# B&R Automation Studio project SW_Shirokov_L2
Automation Studio 4.5.2.102

## Configuration SampleText

### Task classes (Cpu.sw)
```
Cyclic#1 (cycle 2000 us, tolerance 0 us):
  ncsdcctrl <- ncsdcctrl.prg
Cyclic#4:
  Program <- Program.prg
NcDataObjects: acp10etxen <- acp10etxen.dob, gAxis01a <- gAxis01obj.gAxis01a.dob, gAxis01i <- gAxis01obj.gAxis01i.dob
Libraries: Acp10sdc, sys_lib, Runtime, asstring, Library, Acp10man, Acp10par, NcGlobal, Acp10_MC, brsystem, AsBrStr
```

### Hardware
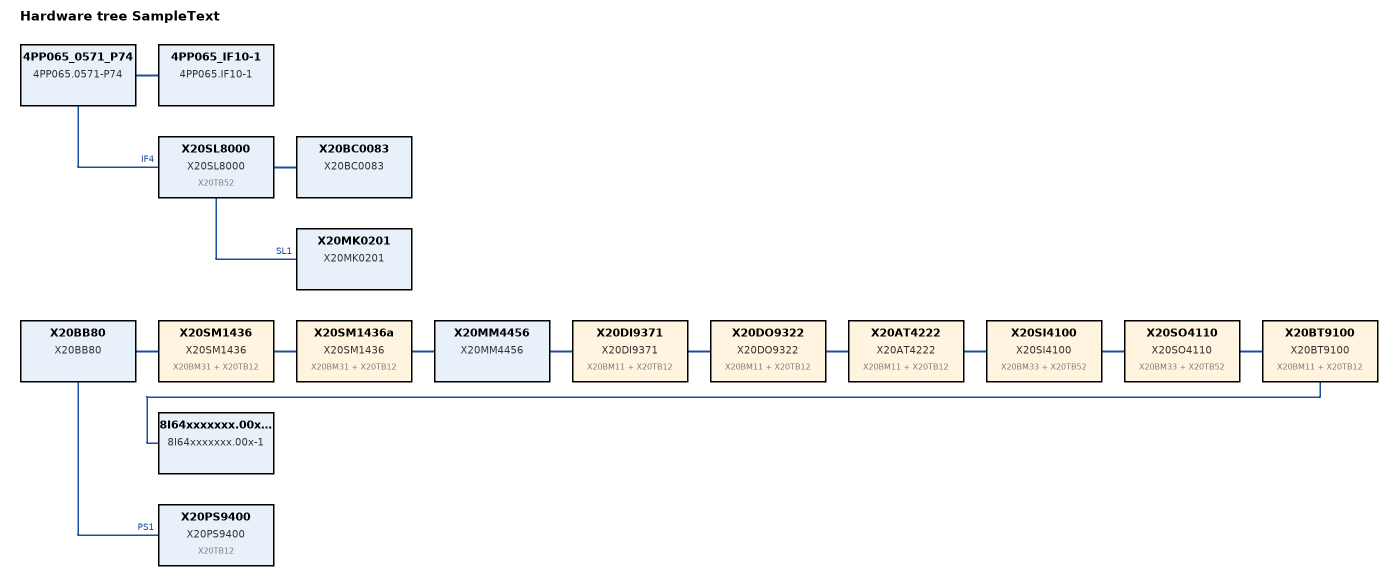
```
4PP065_0571_P74 : 4PP065.0571-P74 v1.1.2.0
  Connector IF5:
    ActivateDevice = 1
    Mode = Manual
    InternetAddress = 10.0.1.10
    SubnetMask = 255.255.255.0
  ConfigurationID = labBR
  TimerDeviceType = EPLX2X
  TimerDevice = 4PP065_0571_P74.IF4
  TaskClassIdleTime = 2000
  Cyclic1Duration = 2000
  Cyclic1Tolerance = 0
  Cyclic1Output = 1
4PP065_IF10-1 : 4PP065.IF10-1 v1.0.3.0  [SS -> 4PP065_0571_P74.SS1]
8I64xxxxxxx.00x-1 : 8I64xxxxxxx.00x-1 v1.3.9.1  [X2X1 -> X20BT9100.X2X1 [Cable Type=X2XCable, Length=10, Version=1.0.0.2]]
  packedETAD = packed
  packedETI = packed
  packedCMDD = packed
  packedCMI = packed
  ACC = 30
  UNS = 220
  NCR = 10
  NSP = 890
  COS = 64
  RSC = 33000
X20AT4222 : X20AT4222 v1.2.3.0  [SS1 -> X20TB12e.SS; SL -> X20BM11c.SL1]
X20BB80 : X20BB80 v1.0.2.0
X20BC0083 : X20BC0083 v2.14.0.0  [PLK1 -> X20SL8000.PLK2 (NodeNumber=2) [Cable Type=PowerlinkCable, Length=10, Version=1.0.0.2]; SL -> X20BB80.SL1]
X20BM11 : X20BM11 v1.0.0.1  [X2X1 -> X20BM33a.X2X2]
X20BM11a : X20BM11 v1.0.0.1  [X2X1 -> X20MM4456.X2X2]
X20BM11b : X20BM11 v1.0.0.1  [X2X1 -> X20BM11a.X2X2]
X20BM11c : X20BM11 v1.0.0.1  [X2X1 -> X20BM11b.X2X2]
X20BM31 : X20BM31 v1.0.0.1  [X2X1 -> X20BB80.IF1]
X20BM31a : X20BM31 v1.0.0.1  [X2X1 -> X20BM31.X2X2]
X20BM33 : X20BM33 v1.0.0.4  [X2X1 -> X20BM11c.X2X2]
X20BM33a : X20BM33 v1.0.0.4  [X2X1 -> X20BM33.X2X2]
X20BT9100 : X20BT9100 v1.0.3.0  [SS1 -> X20TB12f.SS; SL -> X20BM11.SL1]
X20DI9371 : X20DI9371 v1.0.2.0  [SS1 -> X20TB12c.SS; SL -> X20BM11a.SL1]
X20DO9322 : X20DO9322 v1.0.3.0  [SS1 -> X20TB12d.SS; SL -> X20BM11b.SL1]
X20MK0201 : X20MK0201 v1.0.0.0  [SL -> X20SL8000.SL1]
X20MM4456 : X20MM4456 v1.4.0.0  [X2X1 -> X20BM31a.X2X2]
X20PS9400 : X20PS9400 v1.0.2.4  [SS1 -> X20TB12.SS; PS -> X20BB80.PS1]
X20SI4100 : X20SI4100 v1.10.1.1  [SS1 -> X20TB52.SS; SL -> X20BM33.SL1]
X20SL8000 : X20SL8000 v1.6.5.1  [PLK1 -> 4PP065_0571_P74.IF4 (NodeNumber=1) [Cable Type=PowerlinkCable, Length=10, Version=1.0.0.2]; PLK2 -> X20BC0083.PLK1 (NodeNumber=1) [Cable Type=PowerlinkCable, Length=10, Version=1.0.0.2]; SS1 -> X20TB52b.SS]
  SafeProject = SafeLOGIC-1
X20SM1436 : X20SM1436 v2.3.0.0  [SS1 -> X20TB12a.SS; SL -> X20BM31.SL1]
X20SM1436a : X20SM1436 v2.3.0.0  [SS1 -> X20TB12b.SS; SL -> X20BM31a.SL1]
X20SO4110 : X20SO4110 v1.10.1.1  [SS1 -> X20TB52a.SS; SL -> X20BM33a.SL1]
  SafeModuleID = 3
X20TB12 : X20TB12 v1.0.0.0
X20TB12a : X20TB12 v1.0.0.0
X20TB12b : X20TB12 v1.0.0.0
X20TB12c : X20TB12 v1.0.0.0
X20TB12d : X20TB12 v1.0.0.0
X20TB12e : X20TB12 v1.0.0.0
X20TB12f : X20TB12 v1.0.0.0
X20TB52 : X20TB52 v1.0.0.1
X20TB52a : X20TB52 v1.0.0.1
X20TB52b : X20TB52 v1.0.0.1
```

### IoMap.iom - 4PP065_0571_P74/IoMap.iom
```iecst
VAR_CONFIG
	Cyclic#1.gAxis01_DrvIf.iLifeCnt AT %IB."8I64xxxxxxx.00x-1".SDC_LifeCnt;
	Cyclic#1.gAxis01_DrvIf.iDrvOK AT %IX."8I64xxxxxxx.00x-1".ETAD_Input_Bool_02;
	Cyclic#1.gAxis01_DrvIf.oSetTime AT %QW."8I64xxxxxxx.00x-1".SDC_SetTime;
	Cyclic#1.gAxis01_DiDoIf.iLifeCntDriveReady AT %IB."8I64xxxxxxx.00x-1".SDC_LifeCnt;
	Cyclic#1.gAxis01_DiDoIf.iLifeCntDriveEnable AT %IB."8I64xxxxxxx.00x-1".SDC_LifeCnt;
	Cyclic#1.gAxis01_DiDoIf.oDriveEnable AT %QX."8I64xxxxxxx.00x-1".CMDD_Output_Bool_00;
	Cyclic#1.gAxis01_ModuleOk AT %QX."8I64xxxxxxx.00x-1".CMDD_Output_Bool_01;
	Cyclic#1.gAxis01_ModuleOk AT %QX."8I64xxxxxxx.00x-1".CMDD_Output_Bool_02;
	Cyclic#1.gAxis01_ModuleOk AT %IX."8I64xxxxxxx.00x-1".ModuleOk;
	Cyclic#1.gAxis01_DiDoIf.oDriveEnable AT %QX."8I64xxxxxxx.00x-1".CMDD_Output_Bool_03;
	Cyclic#1.gAxis01_DiDoIf.iDriveReady AT %IX."8I64xxxxxxx.00x-1".ETAD_Input_Bool_02;
	::Program:driveSM.state AT %IW."8I64xxxxxxx.00x-1".ETAD_Input;
	::Program:driveSM.command AT %QW."8I64xxxxxxx.00x-1".CMDD_Output;
	::Program:driveSM.speed AT %QW."8I64xxxxxxx.00x-1".LFRD_Output;
	::Program:doorSM.direction AT %IX."X20DI9371".DigitalInput01;
	::Program:doorSM.sw1 AT %IX."X20DI9371".DigitalInput02;
	::Program:doorSM.sw2 AT %IX."X20DI9371".DigitalInput03;
	::Program:doorSM.sw3 AT %IX."X20DI9371".DigitalInput04;
	::Program:doorSM.sw4 AT %IX."X20DI9371".DigitalInput05;
	::Program:ledSM.led1 AT %QX."X20DO9322".DigitalOutput02;
	::Program:ledSM.led2 AT %QX."X20DO9322".DigitalOutput03;
	::Program:ledSM.led3 AT %QX."X20DO9322".DigitalOutput04;
	::Program:ledSM.led4 AT %QX."X20DO9322".DigitalOutput05;
END_VAR
```

## Logical view

Binary libraries used (declarations not repeated): Runtime, Operator, AsIecCon, astime, sys_lib, asstring, Acp10man, Acp10par, NcGlobal, Acp10sdc, Acp10_MC, brsystem, AsBrStr


### Program Logical/Program (ANSIC)

#### Variables.var
```iecst
VAR
	driveSM : {REDUND_UNREPLICABLE} DriveStateMachine := (0);
	ledSM : {REDUND_UNREPLICABLE} LedStateMachine := (0);
	doorSM : {REDUND_UNREPLICABLE} DoorStateMachine := (0);
END_VAR
```

### Library Logical/Library (ANSIC)

#### Types.typ - Exported data types
```iecst
TYPE
	DoorState :
		(
		ST_INIT,
		ST_UNKNOWN,
		ST_OPEN,
		ST_CLOSE,
		ST_ACC_POS,
		ST_ACC_NEG,
		ST_POS,
		ST_NEG,
		ST_DEC_POS,
		ST_DEC_NEG
		);
END_TYPE
```

#### Constants.var - Exported constants
```iecst
VAR CONSTANT
	CMD_ENABLE : UINT := 15;
	CMD_SWITCH_ON : UINT := 7;
	CMD_SHUTDOWN : UINT := 6;
	STATE_DISABLED : UINT := 64;
	STATE_SWITCHED_ON : UINT := 35;
	STATE_READY : UINT := 33;
END_VAR
```

#### Library.fun - Exported functions and function blocks
```iecst
{REDUND_ERROR} {REDUND_UNREPLICABLE} FUNCTION_BLOCK DriveStateMachine (*TODO: Add your comment here*) (*$GROUP=User,$CAT=User,$GROUPICON=User.png,$CATICON=User.png*)
	VAR_INPUT
		state : {REDUND_UNREPLICABLE} UINT;
		enable : {REDUND_UNREPLICABLE} BOOL;
	END_VAR
	VAR_OUTPUT
		command : {REDUND_UNREPLICABLE} UINT;
		speed : {REDUND_UNREPLICABLE} INT;
	END_VAR
	VAR
		mask : {REDUND_UNREPLICABLE} UINT;
	END_VAR
END_FUNCTION_BLOCK

{REDUND_ERROR} {REDUND_UNREPLICABLE} FUNCTION_BLOCK DoorStateMachine (*TODO: Add your comment here*) (*$GROUP=User,$CAT=User,$GROUPICON=User.png,$CATICON=User.png*)
	VAR_INPUT
		state : {REDUND_UNREPLICABLE} UINT;
		sw1 : {REDUND_UNREPLICABLE} BOOL;
		sw2 : {REDUND_UNREPLICABLE} BOOL;
		sw3 : {REDUND_UNREPLICABLE} BOOL;
		sw4 : {REDUND_UNREPLICABLE} BOOL;
		direction : {REDUND_UNREPLICABLE} BOOL;
	END_VAR
	VAR_OUTPUT
		speed : {REDUND_UNREPLICABLE} INT;
	END_VAR
	VAR
		swo1 : {REDUND_UNREPLICABLE} USINT;
		swo2 : {REDUND_UNREPLICABLE} USINT;
		swo3 : {REDUND_UNREPLICABLE} USINT;
		swo4 : {REDUND_UNREPLICABLE} USINT;
	END_VAR
END_FUNCTION_BLOCK

{REDUND_ERROR} {REDUND_UNREPLICABLE} FUNCTION_BLOCK LedStateMachine (*TODO: Add your comment here*) (*$GROUP=User,$CAT=User,$GROUPICON=User.png,$CATICON=User.png*)
	VAR_INPUT
		state : {REDUND_UNREPLICABLE} UINT;
	END_VAR
	VAR_OUTPUT
		led1 : {REDUND_UNREPLICABLE} BOOL;
		led2 : {REDUND_UNREPLICABLE} BOOL;
		led3 : {REDUND_UNREPLICABLE} BOOL;
		led4 : {REDUND_UNREPLICABLE} BOOL;
		timer : {REDUND_UNREPLICABLE} INT;
	END_VAR
END_FUNCTION_BLOCK
```

#### DriveStateMachine.c
```c
#include <bur/plctypes.h>
#ifdef __cplusplus
	extern "C"
	{
#endif
	#include "Library.h"
#ifdef __cplusplus
	};
#endif
/* TODO: Add your comment here */
void DriveStateMachine(struct DriveStateMachine* inst)
{
	/*TODO: Add your code here*/
	mask = inst->state & 0x6f;
	if(!inst->enable)
	{
		inst->command = CMD_SHUTDOWN;
	}
	else
	{
		switch (mask)
		{
			case STATE_DISABLED:
				inst->command = CMD_SHUTDOWN;
				break;

			case STATE_READY:
				inst->command = CMD_ENABLE;
				break;

			case STATE_SWITCHED_ON:
				inst->command = CMD_SWITCH_ON;
				break;
		}
	}
}
```

#### DoorStateMachine.c
```c
#include <bur/plctypes.h>
#ifdef __cplusplus
	extern "C"
	{
#endif
	#include "Library.h"
#ifdef __cplusplus
	};
#endif
/* TODO: Add your comment here */
void DoorStateMachine(struct DoorStateMachine* inst)
{
	/*TODO: Add your code here*/
	switch(inst->state)
	{
		case ST_INIT:
			{
				//if(inst->sw1 == 0 && inst->sw2 == 0 && inst->sw3 == 0 && inst->sw4 == 0) {
				inst->state = ST_UNKNOWN;
				//}
				break;
			}

		case ST_UNKNOWN:
			{
				if(inst->direction == 0 && inst->sw1 != inst->swo1) { //s1=s0?
					inst->state = ST_OPEN;
				}
				if (inst->direction == 1 && inst->sw4 != inst->swo4) { //s3=s2, s4=s3, here s4?
					inst->state = ST_CLOSE;
				}
				break;
			}

		case ST_OPEN:
			{
				inst->speed = 0;
				if(inst->direction == 0) {
					inst->state=ST_ACC_POS;
				}
				break;
			}

		case ST_ACC_POS:
			{
				inst->speed = 250;
				if(inst->sw2 != inst->swo2) { //s2=s1? here s2?
					inst->state = ST_POS;
				}
				if (inst->direction == 1) {
					inst->state = ST_DEC_NEG;
				}
				break;
			}

		case ST_POS:
			{
				inst->speed = 800;
				if(inst->sw3 != inst->swo3) {
					inst->state = ST_DEC_POS;
				}
				if(inst->direction == 1) {
					inst->state = ST_NEG;
				}
			}
			break;

		case ST_DEC_POS:
			{
				inst->speed = 250;
				if(inst->sw4 != inst->swo4) {
					inst->state = ST_CLOSE;
				}
				break;
			}

		case ST_CLOSE:
			{
				inst->speed = 0;
				if(inst->direction == 1) {
					inst->state=ST_ACC_NEG;
				}
				break;
			}

		case ST_ACC_NEG:
			{
				inst->speed = -250;
				if(inst->sw3 != inst->swo3) {
					inst->state = ST_NEG;
				}
				if (inst->direction == 0) {
					inst->state = ST_DEC_POS;
				}
				break;
			}

		case ST_NEG:
			{
				inst->speed = -800;
				if(inst->sw2 != inst->swo2) {
					inst->state = ST_DEC_NEG;
				}
				if(inst->direction == 0) {
					inst->state = ST_POS;
				}
				break;
			}

		case ST_DEC_NEG:
			{
				inst->speed = -250;
				if(inst->sw1 != inst->swo1) {
					inst->state = ST_OPEN;
				}
				break;
			}
	}

	inst->swo1=inst->sw1;
	inst->swo2=inst->sw2;
	inst->swo3=inst->sw3;
	inst->swo4=inst->sw4;
}
```

#### LedStateMachine.c
```c
#include <bur/plctypes.h>
#ifdef __cplusplus
	extern "C"
	{
#endif
	#include "Library.h"
#ifdef __cplusplus
	};
#endif
/* TODO: Add your comment here */
void LedStateMachine(struct LedStateMachine* inst)
{
	/*TODO: Add your code here*/
	switch(inst->state)
	{
		case ST_INIT:
			{
				break;
			}
		case ST_UNKNOWN:
			{
				if(inst->timer%11==10)
				{
					inst->led1=!inst->led1;
					inst->led2=!inst->led2;
					inst->led3=!inst->led3;
					inst->led4=!inst->led4;
				}
				break;
			}
		case ST_OPEN:
			{
				inst->led1=0;
				inst->led2=0;
				inst->led3=0;
				inst->led4=0;
				break;
			}
		case ST_ACC_POS:
			{
				inst->led1=1;
				if(inst->timer%11==10)
					inst->led2=!inst->led2;
				inst->led3=0;
				inst->led4=0;
				break;
			}
		case ST_POS:
			{
				inst->led1=1;
				inst->led2=1;
				if(inst->timer%11==10)
					inst->led3=!inst->led3;
				inst->led4=0;
				break;
			}
		case ST_DEC_POS:
			{
				inst->led1=1;
				inst->led2=1;
				inst->led3=1;
				if(inst->timer%11==10)
					inst->led4=!inst->led4;
				break;
			}
		case ST_CLOSE:
			{
				inst->led1=1;
				inst->led2=1;
				inst->led3=1;
				inst->led4=1;
				break;
			}

		case ST_ACC_NEG:
			{
				inst->led1=1;
				inst->led2=1;
				inst->led3=1;
				if(inst->timer%11==10)
					inst->led4=!inst->led4;

				break;
			}
		case ST_NEG:
			{
				inst->led1=1;
				inst->led2=1;
				if(inst->timer%11==10)
					inst->led3=!inst->led3;
				inst->led4=0;
				break;
			}
		case ST_DEC_NEG:
			{
				inst->led1=1;
				if(inst->timer%11==10)
					inst->led2=!inst->led2;
				inst->led3=0;
				inst->led4=0;

				break;
			}
	}
	inst->timer++;
}
```

Listed in the project but not available here: Logical/Global.typ, Logical/Global.var, Logical/ncsdcctrl, Logical/acp10etxen, Logical/gAxis01obj
